Staubli VAL3: cycle_updateLst.pgx

program cycle_updateLst()
  local num i
  local num l_nSize
  local string l_sEvent
begin
  // get the list
  //
  call prog:getSize(l_nSize)
  resize(sProgList,1,l_nSize)
  sProgList=""
  for i=0 to l_nSize-1
    call prog:get(l_sEvent,i)
    // patch for the #program
    sProgList[i]=l_sEvent
  endFor
end
